FUNCTION_BLOCK FB_FactoryIO_AxisAnalog
VAR_INPUT
    Enable      : BOOL;
    TargetPos   : LREAL;
    ActualPos   : LREAL;

    MaxSpeed    : LREAL := 100;
    Tolerance   : LREAL := 1;

    CycleTime   : LREAL := 0.01;
	error : LREAL;
    step  : LREAL;
END_VAR

VAR_OUTPUT
    CmdPos      : LREAL;
    InPosition  : BOOL;
END_VAR


IF NOT Enable THEN
    CmdPos := ActualPos;
    InPosition := FALSE;
    RETURN;
END_IF

CmdPos := TargetPos;
InPosition := (ABS(TargetPos - ActualPos) <= Tolerance);

END_FUNCTION_BLOCK

(* stored: Version 1.1.0.1
   POU FB_FactoryIO_AxisAnalog: Id {5f5d049b-2f23-458d-a143-1f4e3849ddaa}, SpecialFunc None *)
